{attribute 'global_init_slot' := '49992'}
{attribute 'qualified_only'}
// Robot3 Data
VAR_GLOBAL CONSTANT
	// arm gravity parameters
	(*graParam=[ 2.7244*m3 + 2.7244*m4 + 2.7244*m5 + 2.7244*m6 + 9.8*mx2 + 9.8*mx9,
				9.8*my2 + 9.8*my9,
				3.577*m4 + 3.577*m5 + 3.577*m6 + 0.49*m9 + 9.8*mx3 + 9.8*mx8
				1.5827*m4 + 1.5827*m5 + 1.5827*m6 + 9.8*my3 + 9.8*my8 + 9.8*mz4
				mz5-my4,	my5+mz6,  	mx4,   	mx5, 	mx6,   	my6
				preF2,   k2,   preF3,    k3,    preF5   k5]*)
	g_gravityParam :ARRAY[1..2, 1..16] OF REAL := 
		[ 6.1507, -0.0007155225, 3.320086, 0.48504608, -0.03643, 0.02393, 0.0000375, 0.0000117, 0.00008169, -0.0147358, 
			8.7047302, 3101.998, 7.7845, 1989.9943, 1.112, 477.91541,
		  6.3336386, -0.0002385075, 4.3071, 1.060203, -0.043111496, 0.022730322, 0.0000375, 0.0000117, -0.000929, -0.015102275, 
			7.7845, 3195.0, 12.455128, 2842.287, 2.6162855, 454.267];
			
	// gravity deviation
	g_gravityDeviaion :ARRAY[1..2, 1..7] OF REAL :=
	[ 0.0, 0.0, -0.02, 0.0, 0.0025, 0.005, 0.0, 
	 0.0, 0.0, 0.0, 0.0, -0.0025, -0.005, 0.0];
	  
	// arm friction parameters [a1,b1,...a7,b7];
	// friction = a * gravity + b; only joint 5 and 6 is identified
	g_jntFrictionParam :ARRAY[1..2, 1..14] OF LREAL :=
	[ 0, 0.052118501, 0, 0.050075801, 0.02, 0.036312347, 0.101, 0.02608, 0.21596626, 0.012022009, 0.23862478, 0.004035171, 0, 0.004418365,
	  0, 0.063615008, 0.03, 0.055326576, 0.113, 0.062596658, 0.19, 0.018976863, 0.24246004, 0.0083495406, 0.30998273, 0.0053789188, 0, 0.0046038532];
	g_maxJntFriction : Vec7d :=[0.2, 0.2, 0.2, 0.1, 0.1, 0.1, 0.01];
	
	//################ dynamic reference model parameters below ###########################
	// link mass [m1, m2, m3, m4, m5, m6, m7, m8, m9]
	g_linkMass :ARRAY[1..9] OF LREAL :=[2.676, 0.825, 0.547, 0.25, 0.195, 0.194, 0.05, 0.111, 0.09] ;
	
	// lin center of amss
	g_linkCOM :ARRAY[1..9,1..3] OF LREAL := [   1.376E-3,    -1.019E-3,  -81.464E-3,
										   90.622E-3,   -0.113E-3,  15.088E-3,
										   167.4E-3,    3.7E-3,     -0.438E-3,
										   0.1E-3,      98.49E-3,   -55.74E-3,
										   0.12E-3,     76.667E-3,  -36E-3,
										   0,           -61.63E-3,  27.3E-3,
										   0.06E-3,     -0.08E-3,   17.671E-3,
										   11E-3,       -3.364E-3,  39.265E-3,
										   143e-3,      0.495e-3,   24.253e-3];
	// link  inertial
    // [Ixx,Iyy,Izz, Ixy,Ixz, Iyz]
 	g_linkInertia :ARRAY[1..9,1..6] OF LREAL :=[  19.63E-3,   16.43E-3,  12.7E-3,   -0.3222E-3,    -0.667E-3,     -0.0268E-3,
												   1.017E-3,   6.637E-3,  5.935E-3,  -0.037E-3,     -0.238E-3,     0.06E-3,
												   0.161E-3,   9.572E-3,  9.586E-3,  0.0447E-3,     0.0277E-3,     0.465E-6,
												   0.992E-3,   0.707E-3,  0.335E-3,  0.2E-6,     2E-6,       0.224E-3,
												   0.402E-3,   0.25E-3,   0.186E-3,  0.002E-6,   -1.2E-6,    0.106E-3,
												   0.281E-3,   0.178E-3,  0.137E-3,  0.076E-6,   0.09E-6,    0.056E-3,
												   0.0255E-3,  0.0259E-3, 5.96E-6,0.34E-6,    -3E-9,      24E-9,
												   0.033E-3,   0.0976E-3, 0.126E-3,  3E-6,       -5E-6,      -0.162E-6,
												   4.9E-6,  0.757E-3,  0.760E-3,  2.6E-6,     -5.3E-6,    -18E-9];

	//################ DO NOT modify parameters below ###########################
	//  motor inertial at link size
	g_motorInertia :ARRAY[1..7] OF LREAL := [34.7E-7, 34.7E-7, 34.7E-7, 9.26E-7, 0.495E-7, 0.495E-7, 0.495E-7];
	
	// spring parameters
	// spring2 [L0, b1, b2, l1, r0]
	g_spring2Param :ARRAY[1..5] OF LREAL :=[101.6E-3, 14.5E-3, 15E-3, 172E-3, 31E-3];
	// spring3 [L0, b1, b2, l1, r0,d]
	g_spring3Param :ARRAY[1..6] OF LREAL :=[101.6E-3, 14E-3, 15E-3, 172E-3, 30E-3, 10E-3];
	// spring5 [L0, s1, L1, r0, beta]
	g_spring5Param :ARRAY[1..5] OF LREAL :=[34.93E-3, 34.3E-3, 100E-3, 12.5E-3, 32.02*g_deg2rad];
	
END_VAR

(* stored: Version 1.1.0.1, ProductVersion 3.1.4024.12
   GVL GVL_ArmDynamics_3: Id {9220a6fd-c631-4b1f-926c-9e28ee7c87ad} *)
